// FB_UnitBase suite: mode rejection, run-as-command, stall key, wait-class
// derived Starved, cycle publication, mode change = immediate software abort by default.
FUNCTION_BLOCK FB_Unit_Tests EXTENDS TcUnit.FB_TestSuite
VAR
    _u : FB_ProbeUnit;
    _w : BOOL;
    _wCfg : BOOL;
    _pager : FB_ConfigPager;
    _page : ST_ConfigPage;
END_VAR

Unit_run_stall_classes_and_cycle();
Unit_mode_change_is_estop_by_default();
Sequence_rows_belong_to_the_active_mode();
Unit_config_capability_is_typed_and_fail_closed();

METHOD Unit_run_stall_classes_and_cycle
TEST('Unit_run_stall_classes_and_cycle');
IF NOT _w THEN
    _u.Setup('Test.Unit');
    _w := TRUE;
END_IF
AssertFalse(Condition := _u.SetMode(Mode := E_Mode.CALIBRATION),
            Message := 'unsupported mode rejected gracefully (3.4/3.7)');
AssertTrue(Condition := _u.Start(), Message := 'Start issues the run command (6 intro)');
_u();                                         // edge -> BUSY, step 100 set
_u();                                         // stall guard (T#0S) fires -> pending
AssertTrue(Condition := _u.Busy, Message := 'running');
AssertEquals_DWORD(Expected := TO_DWORD(E_Reason.STEP_STALLED),
                   Actual   := TO_DWORD(_u.Pending.ReasonCode),
                   Message  := 'stall is a PENDING reason, not a fault (6.9)');
AssertEquals_STRING(Expected := 'std.diagnostic.stepStalled',
                    Actual   := _u.Pending.Description,
                    Message  := 'stall publishes a stable key; CurrentStep carries context');
AssertFalse(Condition := _u.Error, Message := 'no fault from a stall');
_u.SimA := TRUE;
_u();                                         // -> step 200 (WAIT_UPSTREAM)
_u();
AssertTrue(Condition := _u.Starved,
           Message := 'Starved derived from the step wait class (8.11.4f/8.11.3)');
_u.Stop();
_u.SimB := TRUE;
_u();                                         // -> step 30
_u();                                         // EndOfCycle: publish + complete + release
_u();                                         // reset -> READY
AssertFalse(Condition := _u.Busy, Message := 'stopped after cycle (3.3)');
AssertEquals_INT(Expected := 2, Actual := _u.Profiler.LastCycle.NSteps,
                 Message := 'cycle profile published with both steps (8.11.4b)');
TEST_FINISHED();
END_METHOD

METHOD Unit_config_capability_is_typed_and_fail_closed
VAR
    i : INT;
    found : BOOL;
    pageIndex : INT;
    pageCount : INT;
END_VAR
TEST('Unit_config_capability_is_typed_and_fail_closed');
// Latched like the stall test above it. Without this the method re-ran every
// scan against a Unit that test leaves BUSY, and the READY-gated write below
// was then refused CORRECTLY - so the failure measured the mode gate rather
// than the capability it names.
IF NOT _wCfg THEN
_wCfg := TRUE;
// The capability publishes RequiresReady, so put the Unit where that is true.
_u.Stop();
FOR i := 1 TO 10 DO
    _u();
END_FOR
AssertFalse(Condition := _u.Busy,
    Message := 'the Unit is idle before a READY-gated write is attempted');
found := FALSE;
_pager.M_Setup(Target := ADR(_page), PageIndex := 0, Revision := 1);
_u.M_AppendConfig(Pager := _pager);
_pager.M_Finish();
pageCount := _page.PageCount;
// The manifest is a bounded window. Search every advertised page instead of
// coupling this contract test to the current number/order of base entries.
FOR pageIndex := 0 TO pageCount - 1 DO
    _pager.M_Setup(Target := ADR(_page), PageIndex := pageIndex, Revision := 1);
    _u.M_AppendConfig(Pager := _pager);
    _pager.M_Finish();
    FOR i := 1 TO _page.EntryCount DO
        IF _page.Entries[i].WriteKey = 'unit.modePolicy.3.shield' THEN
            found := TRUE;
            AssertTrue(Condition := _page.Entries[i].Writable,
                Message := 'mode policy is an explicit write capability');
            AssertEquals_UDINT(Expected := 1, Actual := _page.Entries[i].WriteRevision,
                Message := 'write capability has a non-zero schema revision');
            AssertTrue(Condition := _page.Entries[i].RequiresReady,
                Message := 'capability publishes its READY-state constraint');
        END_IF
    END_FOR
END_FOR
AssertTrue(Condition := found, Message := 'stable mode-policy key is manifest-served');
AssertTrue(Condition := _u.WriteConfig(TargetPath := 'Test.Unit',
    WriteKey := 'unit.modePolicy.3.shield', Revision := 1, TextValue := '0'),
    Message := 'registered exact enum value is accepted while READY');
AssertEquals_DINT(Expected := TO_DINT(E_ModeSwitchShield.INTERRUPTIBLE),
    Actual := TO_DINT(_u.ModePolicy[3].Shield), Message := 'typed handler applied value');
AssertFalse(Condition := _u.WriteConfig(TargetPath := 'Test.Unit',
    WriteKey := 'unit.modePolicy.3.shield', Revision := 2, TextValue := '1'),
    Message := 'stale capability revision is rejected');
AssertFalse(Condition := _u.WriteConfig(TargetPath := 'Test.Unit',
    WriteKey := 'unit.modePolicy.3.shield', Revision := 1, TextValue := '9'),
    Message := 'out-of-domain value is rejected');
AssertFalse(Condition := _u.WriteConfig(TargetPath := 'Other.Unit',
    WriteKey := 'unit.modePolicy.3.shield', Revision := 1, TextValue := '1'),
    Message := 'foreign owner path is rejected');
END_IF
TEST_FINISHED();
END_METHOD

METHOD Sequence_rows_belong_to_the_active_mode
TEST('Sequence_rows_belong_to_the_active_mode');
// The previous test left the Unit in MANUAL having run two AUTO steps, so the §3.13
// table had rows in it when the mode committed. Discovery has no end of its own:
// without a boundary the chart becomes the union of every chain run since boot.
AssertEquals_INT(Expected := 0, Actual := _u.SequenceStepCount,
    Message := 'committing a mode drops the previous mode chain rows');
AssertEquals_INT(Expected := 0, Actual := _u.SequenceStepDef[1].StepNo,
    Message := 'and clears them, so a later row cannot inherit stale text');
// the new mode fills its own table from scratch
AssertTrue(Condition := _u.SetMode(Mode := E_Mode.AUTO), Message := 'back to AUTO');
_u();
_u();
_u();
AssertTrue(Condition := _u.Start(), Message := 'run the AUTO chain again');
_u();
AssertEquals_INT(Expected := 1, Actual := _u.SequenceStepCount,
    Message := 'the chart rebuilds from the mode that is actually running');
TEST_FINISHED();
END_METHOD

METHOD Unit_mode_change_is_estop_by_default
TEST('Unit_mode_change_is_estop_by_default');
_u.SimA := FALSE;
_u.SimB := FALSE;
AssertTrue(Condition := _u.Start(), Message := 're-start');
_u();
AssertTrue(Condition := _u.Busy, Message := 'running again');
AssertTrue(Condition := _u.SetMode(Mode := E_Mode.MANUAL), Message := 'mode request accepted (pending)');
_u();                                         // OnModeExit=0 -> OnAbort (non-safety software abort, 3.14.4)
_u();                                         // release run command, reset
_u();                                         // commit mode
AssertFalse(Condition := _u.Busy, Message := 'chain cancelled by the mode change');
AssertEquals_UDINT(Expected := 1, Actual := _u.ModeExitCount,
    Message := 'OnModeExit runs once for this immediate transition');
AssertEquals_UDINT(Expected := 1, Actual := _u.ModeExitFirstCount,
    Message := 'OnModeExit receives FirstCall exactly once');
AssertEquals_DINT(Expected := TO_DINT(E_Mode.MANUAL),
    Actual := TO_DINT(_u.LastRequestedMode),
    Message := 'OnModeExit receives the pending target mode');
AssertEquals_UDINT(Expected := 1, Actual := _u.ModeChangedCount,
    Message := 'OnModeChanged runs once after commit');
AssertEquals_DINT(Expected := TO_DINT(E_Mode.AUTO),
    Actual := TO_DINT(_u.LastOldMode),
    Message := 'OnModeChanged receives the mode being left');
AssertEquals_DINT(Expected := TO_DINT(E_Mode.MANUAL),
    Actual := TO_DINT(_u.LastNewMode),
    Message := 'OnModeChanged receives the committed mode');
AssertEquals_DINT(Expected := TO_DINT(E_Mode.MANUAL),
                  Actual   := TO_DINT(_u.ModeActive),
                  Message  := 'mode committed after leaving BUSY (3.14.4)');
AssertEquals_DINT(Expected := TO_DINT(E_HostEventKind.MODE_CHANGED),
    Actual := TO_DINT(_u.HostEvents.Ring[_u.HostEvents.RingHead].Kind),
    Message := 'base emits the fixed mode host event once committed');
AssertEquals_STRING(Expected := 'Test.Unit',
    Actual := _u.HostEvents.Ring[_u.HostEvents.RingHead].StationPath,
    Message := 'host event owns the qualified root path');
AssertEquals_STRING(Expected := '1',
    Actual := _u.HostEvents.Ring[_u.HostEvents.RingHead].Value,
    Message := 'new mode is projected in the compact event value');
TEST_FINISHED();
END_METHOD

END_FUNCTION_BLOCK

(* stored: Version 1.1.0.1, ProductVersion 3.1.4024.12
   POU FB_Unit_Tests: Id {ccffa0fb-4bf8-45f8-837f-baf7462dfa55}, SpecialFunc None
   Method Unit_run_stall_classes_and_cycle: Id {14ae51c7-c760-4004-9fdd-4ede7d4f00ff}
   Method Unit_config_capability_is_typed_and_fail_closed: Id {733c367d-063e-43d5-bcc8-d27e71a9182a}
   Method Sequence_rows_belong_to_the_active_mode: Id {02a7b2be-5959-445e-aa14-e646770d0bdd}
   Method Unit_mode_change_is_estop_by_default: Id {7c014f2f-fda2-494e-b29c-1fc8224ac0ab} *)
